FUNCTION Convert_TOD_TO_LREAL : Hresult
VAR_INPUT
	in : TOD;
	out : REFERENCE TO LREAL;
END_VAR
VAR
	converted : LREAL;
END_VAR
VAR CONSTANT
	INCOMPATIBLE : HRESULT := 16#9811070E;
END_VAR

converted := TOD_TO_LREAL(in);

IF (LREAL_TO_TOD(converted) <> in) THEN
	Convert_TOD_TO_LREAL := INCOMPATIBLE;
	RETURN;
END_IF

out := converted;

END_FUNCTION

(* stored: Version 1.1.0.1, ProductVersion 3.1.4024.12
   POU Convert_TOD_TO_LREAL: Id {179b569b-1787-45d9-8976-e8c04de27bb7}, SpecialFunc None *)
